TYPE ServicesTimingPositionSource :
(
	CONFIG := 0,
	GPS := 1
);
END_TYPE

(* stored: Version 1.1.0.1, ProductVersion 3.1.4018.5
   DUT ServicesTimingPositionSource: Id {591b46fc-3e6e-4de1-a038-8b3f536ee6bd} *)
